Universal Robots PolyScope program: hello_world_script.urp

Program hello_world_script (installation=default directory=/home/hugo/Documents/Proyecto_Ingenieria/ursim-5.10.2.106319/programs/ASM createdIn=5.10.2.106319 lastSavedIn=5.10.2.106319 robotSerialNumber=20195599999)
Calibrated DH parameters: a=[0, -0.425, -0.3922, 0, 0, 0]; d=[0.1625, 0, 0, 0.1333, 0.0997, 0.0996]; alpha=[1.570796, 0, 0, 1.570796, -1.570796, 0]; deltaTheta=[0, 0, 0, 0, 0, 0]
Robot Program (runOnlyOnce=false)
  Script file /home/hugo/Documents/Proyecto_Ingenieria/ursim-5.10.2.106319/programs/ASM/hola_mundo.script
    | def hola_mundo():
    | 	popup("Hola Mundo", blocking=True)
    | end
    | 
    | def adios_mundo():
    | 	popup("Adios Mundo", blocking=True)
    | end
  Script: hola_mundo()
  Script: adios_mundo()
